// TIA Portal V19 export
DATA_BLOCK "Sensors_DB"   // DB4
// stored: InstanceOfName Sensors, InstanceOfType FB
"Sensors"
   // VAR
   //    GenericSensor11 { S7_SetPoint := 'True'} : "GenericSensor";
   //    GenericSensor12 { S7_SetPoint := 'True'} : "GenericSensor";
   //    GenericSensor13 { S7_SetPoint := 'True'} : "GenericSensor";
   //    GenericSensor21 { S7_SetPoint := 'True'} : "GenericSensor";
   //    GenericSensor22 { S7_SetPoint := 'True'} : "GenericSensor";
   //    PubJsonMqttInst11 { S7_SetPoint := 'True'} : "PublishJsonMqtt";
   //    PubJsonMqttInst12 { S7_SetPoint := 'True'} : "PublishJsonMqtt";
   //    PubJsonMqttInst13 { S7_SetPoint := 'True'} : "PublishJsonMqtt";
   //    PubJsonMqttInst21 { S7_SetPoint := 'True'} : "PublishJsonMqtt";
   //    PubJsonMqttInst22 { S7_SetPoint := 'True'} : "PublishJsonMqtt";
   //    tpGen01 { S7_SetPoint := 'True'} : TP_TIME;
   //    tpGen02 { S7_SetPoint := 'True'} : TP_TIME;
   //    tpGen03 { S7_SetPoint := 'True'} : TP_TIME;
   //    tpGen04 { S7_SetPoint := 'True'} : TP_TIME;
   // END_VAR
BEGIN
END_DATA_BLOCK
